PROGRAM MAIN
VAR
	rReadAnalog1 : REAL;
	rReadAnalog2 : REAL;
END_VAR

rReadAnalog1 := INT_TO_REAL(GVL.Analog_Inputs_Res[1])/32767*10;
rReadAnalog2 := INT_TO_REAL(GVL.Analog_Inputs_Res[2])/32767*10;

END_PROGRAM

(* stored: Version 1.1.0.1, ProductVersion 3.1.4024.12
   POU MAIN: Id {56d10763-6796-48b8-aa8b-e9d8277f85a7}, SpecialFunc None *)
